FUNCTION_BLOCK HaltedToReadyUnifiedProgramTransition EXTENDS HaltedToReadyProgramTransition
VAR
	{attribute 'OPC.UA.DA' := '0'}
	_ClassName : STRING := __POUNAME();
END_VAR

{attribute 'monitoring' := 'call'}
PROPERTY ClassName : STRING
GET
ClassName := _ClassName;
END_GET
END_PROPERTY

END_FUNCTION_BLOCK

(* stored: Version 1.1.0.1
   POU HaltedToReadyUnifiedProgramTransition: Id {12116f2f-f0c0-4f18-8a0b-b696fc4276d9}, SpecialFunc None
   Property ClassName: Id {6039b23e-92d1-4be2-a6f7-b27baffc1eca}
   Get Get: Id {98caf3c1-7a78-4186-924b-8ecc289abfac} *)
